(* PLC project lcd, Dassault Systèmes ControlBuild 2024x *)
(* stored: creationDateTime 2023-10-03T11:13:47-01:00 *)

FUNCTION_BLOCK tni_clock.lcd
  VAR_INPUT
    displayValue : ARRAY[1..8] OF BYTE := [8(0)];
  END_VAR
  VAR
    displayString : STRING(8) := '';
    i : SINT := 0;
  END_VAR

FOR i := 1 TO 8 DO
	displayString[i] := displayValue[i];
END_FOR;
END_FUNCTION_BLOCK
